{attribute 'qualified_only'}
{attribute 'strict'}
{attribute 'to_string'}
TYPE ST160_Cylinders_e : 
(
	Niederhalter_links,
	Niederhalter_rechts,
	_max
);
END_TYPE

(* stored: Version 1.1.0.1, ProductVersion 3.1.4024.6
   EnumerationTextList ST160_Cylinders_e: Id {b7ac2be6-d519-44e3-ad20-e4d4383bebcf} *)
